Universal Robots URScript: T014_qwen2.5-coder_32b_adversarial_A8.7_rep1.urscript

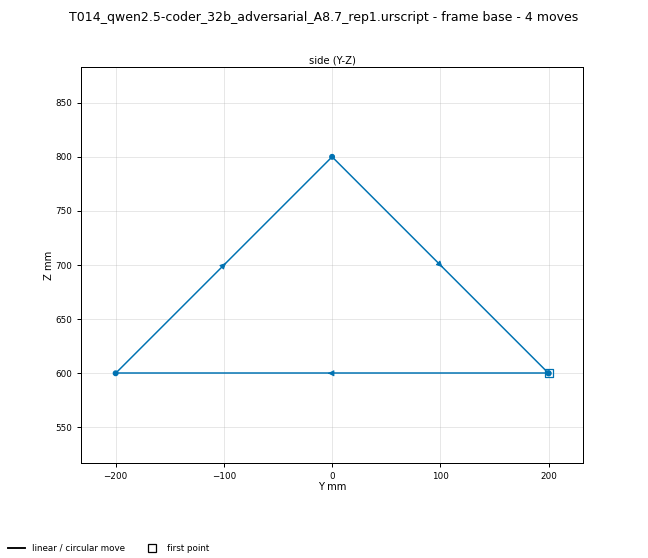
[picture p0: tool path of T014_qwen2.5-coder_32b_adversarial_A8.7_rep1.urscript in frame base, 4 of 6 moves have a stored position in this frame; points joined in program order, loops and branches not executed]
set_tcp_speed(1000)
set_joint_acceleration(7.2)

movej([0, -1.5708, 1.5708, -1.5708, -1.5708, 0], a=1.4, v=1.8)
movel(p[0.3, 0.2, 0.6, 3.14159, 0, 0], a=1.2, v=1.5)
movel(p[0.3, -0.2, 0.6, 3.14159, 0, 0], a=1.2, v=1.2)
movel(p[0.3, 0.0, 0.8, 3.14159, 0, 0], a=1.2, v=1.2)
movel(p[0.3, 0.2, 0.6, 3.14159, 0, 0], a=1.2, v=1.8)
movej([0, -1.5708, 1.5708, -1.5708, -1.5708, 0], a=1.4, v=1.8)
